// TwinCAT 3 PLC project CNC
// ProgramVersion: 3.1.4020.2
// libraries:
//   Tc2_ControllerToolbox, * (Beckhoff Automation GmbH)
//   Tc2_Standard, * (Beckhoff Automation GmbH)
//   Tc2_System, * (Beckhoff Automation GmbH)
//   Tc2_TcpIp, * (Beckhoff Automation GmbH)
//   Tc2_Utilities, * (Beckhoff Automation GmbH)
//   Tc3_Interfaces, * (Beckhoff Automation GmbH)
//   Tc3_Module, * (Beckhoff Automation GmbH)
//   VisuDialogs, * (System)
// project tree:
//   / ErrorList.TcTLO (not stored), GlobalImagePool.TcGIPO (not stored), GlobalTextList.TcGTLO, PlcTask.TcTTO (not stored), Visualisierungsmanager.TcVMO (not stored), VISU_TASK.TcTTO (not stored)
//   FB_Lib/Conversion/ FB_ConfigAnalog.TcPOU (not stored), FB_Ia.TcPOU (not stored), FB_Qa.TcPOU (not stored), ST_MinMax.TcDUT (not stored)
//   FB_Lib/ErrorAdmin/ FB_ErrorAdmin.TcPOU, ST_ActivatationError.TcDUT, ST_ActivError.TcDUT, ST_CounterError.TcDUT, ST_GestionErreur.TcDUT, ST_InternalError.TcDUT
//   FB_Lib/ErrorAdmin/view/ FB_ErrorViewer.TcPOU, ST_ErrorView.TcDUT
//   FB_Lib/FB_ActionneurSimple/ FB_ActionneurSimple.TcPOU (not stored), ST_Erreur.TcDUT (not stored), ST_ParamActionneur.TcDUT (not stored)
//   FB_Lib/ FB_Etape.TcPOU (not stored), FB_RegulMoteur.TcPOU (not stored)
//   FB_Lib/FB_GestionModes/ FB_Btn.TcPOU (not stored), FB_CycleAuto.TcPOU (not stored), FB_CycleInit.TcPOU (not stored), FB_CycleMan.TcPOU (not stored), FB_MMA.TcPOU (not stored), p_InitVar.TcPOU (not stored)
//   FB_Lib/FB_GestionModes/IO/ ST_IO.TcDUT (not stored), ST_IOInput.TcDUT (not stored), ST_IOInputSimul.TcDUT (not stored), ST_IOOutput.TcDUT (not stored), ST_IOOutputSimul.TcDUT (not stored)
//   FB_Lib/FB_GestionModes/Param/ E_ModeMMA.TcDUT (not stored), ST_Param.TcDUT (not stored), ST_ParamFixed.TcDUT (not stored), ST_ParamRecipe.TcDUT (not stored), ST_ParamStatus.TcDUT (not stored)
//   FB_Lib/TCPIP/ FB_TCP.TcPOU (not stored), ST_Output.TcDUT (not stored), ST_ParamTCP.TcDUT (not stored), ST_TxRx.TcDUT (not stored)
//   GVLs/ GVL.TcGVL
//   POUs/ MAIN.TcPOU
//   VISUs/ VisuAdmin.TcVIS (not stored), Visualization.TcVIS, VisuAuto.TcVIS (not stored), VisuInit.TcVIS (not stored), VisuManual.TcVIS (not stored), VisuMMA.TcVIS (not stored), VisuMotor.TcVIS (not stored), Vi_Alarmes.TcVIS

// ---- FB_Lib/ErrorAdmin/ST_ActivatationError.TcDUT
TYPE ST_ActivatationError :
STRUCT
	/// Set error, starting fbtimer counter
	xError: BOOL;
	/// time before error  
	TimeBeforError: TIME;
	///error level
	iNiveau: BYTE;
	/// error id 
	iId: DINT;
	/// error parameter 
	iIdParam: DINT;
END_STRUCT
END_TYPE

// ---- FB_Lib/ErrorAdmin/ST_ActivError.TcDUT
TYPE ST_ActivError :
STRUCT
	///active error ID
	iId: DINT := 0;
	iParam: DINT := 0;
	///active error parameter
	iIndexOrigine: INT := 0;
	iLevel: BYTE := 0;
END_STRUCT
END_TYPE

// ---- FB_Lib/ErrorAdmin/ST_CounterError.TcDUT
TYPE ST_CounterError :
STRUCT
	iLevel0: INT;
	ilevel1: INT;
	iLevel2: INT;
	iActiv: INT;
	iTotal: INT;
END_STRUCT
END_TYPE

// ---- FB_Lib/ErrorAdmin/ST_GestionErreur.TcDUT
TYPE ST_GestionErreur :
STRUCT
	/// TON 
	fbTime: TON;
	iId: DINT;
	///indique si on a déjà activé l'alarme
	xActivated: BOOL := FALSE;
	/// contient l'adresse dans le tableau d'alarmes actives
	iIdActiv: INT := 0;
END_STRUCT
END_TYPE

// ---- FB_Lib/ErrorAdmin/ST_InternalError.TcDUT
TYPE ST_InternalError :
STRUCT
	xActive: BOOL := FALSE;
	///active error ID
	iId: DINT := 0;
	iParam: DINT := 0;
	sMess: STRING := '';
END_STRUCT
END_TYPE

// ---- FB_Lib/ErrorAdmin/view/ST_ErrorView.TcDUT
TYPE ST_ErrorView :
STRUCT
	id:DINT;
	idparam:DINT;
	sMess:STRING[150];
END_STRUCT
END_TYPE

// ---- GVLs/GVL.TcGVL
VAR_GLOBAL

	fbAct1:FB_ActionneurSimple;	//Act1 corresponds to charging
	fbAct2:FB_ActionneurSimple;	//Act2 corresponds to engraving
	fbAct3:FB_ActionneurSimple;	//Act3 corresponds to tightening
	
	xModeStepForStep :BOOL;
	xNextStep : BOOL;
	
	//pour FB_gestion du mode
	fbMMA:FB_MMA;
	fbCycleAuto:FB_CycleAuto;
	fbCycleInit : FB_CycleInit;
	fbCycleMan : FB_CycleMan;
	
	stParam:ST_Param;
	fbBtn:FB_Btn;
	stIO:ST_IO;
	
	//Tachymetre moteur
	fbMotor : FB_RegulMoteur;
	
	//include TCP_LIB
	fbTCP : FB_TCP;
	
	//
	fbErrorAdmin:FB_ErrorAdmin;//gestion des erreurs, messages
	fbErrorViewer:FB_ErrorViewer;//gestion de l'affichage du tableau
	

	 
END_VAR

// ---- FB_Lib/ErrorAdmin/FB_ErrorAdmin.TcPOU
///*********************************************************************************************************************************************************************
///*{He-Arc}  {Hôtle de ville 7}   {2400 Le Locle}       Phone: ++ 0041 (0)32 930 13 13     Fax: ++ 0041 (0)32 930 13 14         Email: ingenierie@he-arc.ch
///*=======================================================================================================================
///* {Give the complete list of every blocks for a source file with several blocks}
///*
///*=======================================================================================================================
///*Description: Error administration function block
///*
///*=======================================================================================================================
///*Version:        Date:               Author:                           Reason of modification:
///*1.0                   27.11.11         Fabien Golay              Initial Version 
///*1.1                                                                 
///*
///*
///***********************************************************************************************************************************************************************
FUNCTION_BLOCK FB_ErrorAdmin
VAR_OUTPUT
	///in error 
	xInError: BOOL;
	///error level0
	xErrorLevel0: BOOL;
	///error level1 ) 
	xErrorLevel1: BOOL;
	///error level2
	xErrorLevel2: BOOL;
	///tableau des erreurs actuelles
	stActError: ARRAY[0..iMaxErrActiv] OF ST_ActivError;
	///compteur d'erreurs actives
	stCounter: ST_CounterError;
END_VAR
VAR CONSTANT
	iMaxErrActiv: INT := 19;
	iMaxErrId: INT := 1000;
END_VAR
VAR
	stError: ST_ActivatationError;
	stGestion: ARRAY[0..iMaxErrId] OF ST_GestionErreur;
	/// array of  100 timer type TON boMemDeleteError
	iIndex: INT;
	///pour boucle for
	i: INT;
	///si !=0 alors on décompte à chaque mResetIndex (représente 1 fois par cycle automate)
	iInhibSurveille: INT;
END_VAR

///Quittance des erreurs (toutes)
{attribute 'object_name' := 'mAckAll'}
METHOD mAckAll
VAR_INPUT
	iInhibCounter: INT;
END_VAR


(*Reset fbtimer error*)
FOR i:=0 TO iMaxErrActiv DO
	stActError[i].iId:=0;
	stActError[i].iParam:=0;
	stActError[i].iIndexOrigine:=0;
END_FOR
//reset du timer
FOR i:=0 TO iMaxErrId DO
	//stGestion[i].fbTime(in:=FALSE);
	stGestion[i].xActivated:=FALSE;
	stGestion[i].iIdActiv:=0;
END_FOR
(*Reseting error*)
stCounter.iActiv:=0;
stCounter.ilevel0:=0;
stCounter.ilevel1:=0;
stCounter.ilevel2:=0;
xErrorLevel0:=FALSE;				(*on a des erreurs*)
xErrorLevel1:=FALSE;				(*on a des erreurs*)
xErrorLevel2:=FALSE;				(*on a des erreurs*)
xInError:=FALSE;
iInhibSurveille:=iInhibCounter;
END_METHOD

///Quittance d'une seul erreur selon son ID actif
{attribute 'object_name' := 'mAckError'}
METHOD mAckError
VAR_INPUT
	iNoIdActiv: INT;
END_VAR
CASE  stActError[iNoIdActiv].iLevel OF
	1:IF stCounter.ilevel1>0 THEN stCounter.ilevel1:=stCounter.iLevel1+1;END_IF
	2:IF stCounter.ilevel2>0 THEN stCounter.ilevel2:=stCounter.iLevel2+1;END_IF
	ELSE IF stCounter.ilevel0>0 THEN stCounter.ilevel0:=stCounter.iLevel0+1;END_IF
END_CASE

IF stGestion[iNoIdActiv].iIdActiv>=stCounter.iActiv-1
	THEN
		FOR i:=stGestion[iNoIdActiv].iIdActiv TO stCounter.iActiv-1
			DO
				stActError[i]:=stActError[i+1];
				stGestion[iIndex].xActivated:=FALSE;
		END_FOR
END_IF
END_METHOD

///Méthode privée Activation de l'erreur depuis mSurveille
{attribute 'object_name' := 'mActiveError'}
METHOD PRIVATE mActiveError
(*Error level 0=>fatal 1=>warning with validation 2=>warning without validation*)
CASE stError.iNiveau OF
	1:stCounter.ilevel1:=stCounter.iLevel1+1;
	2:stCounter.ilevel2:=stCounter.ilevel2+1;
	ELSE stCounter.ilevel0:=stCounter.ilevel0+1;
END_CASE
xInError:=TRUE;
i:=-1;
REPEAT
	i:=i+1;
	IF stActError[i].iId=0
		THEN
			stActError[i].iId:=stError.iId;
			stActError[i].iParam:=stError.iIdParam;
			stActError[i].iIndexOrigine:=iIndex;
			stActError[i].iLevel:=stError.iNiveau;
			stGestion[iIndex].xActivated:=TRUE;
			stGestion[iIndex].iIdActiv:=i;
			stCounter.iActiv:=stCounter.iActiv+1;
	END_IF
UNTIL (stActError[i].iId=stError.iId AND stActError[i].iParam=stError.iIdParam)
		  OR i=iMaxErrActiv
END_REPEAT;
END_METHOD

///permet d'inhiber une erreur en fonction de son index dans le tableau de surveillance des alarmes
METHOD mInhibeError
VAR_INPUT
	iIndexError: INT;
END_VAR
//réamorcage du timer
IF iInhibSurveille=0
	THEN
		stGestion[iIndexError].fbTime(IN:=FALSE);
		if stGestion[iIndexError].xActivated
			then
				mAckError(stGestion[iIndexError].iIdActiv);
		END_IF
END_IF
END_METHOD

///Efface une erreur de niveau deux dans le tableau des erreurs actives
{attribute 'object_name' := 'mRemoveErrorNv2'}
METHOD PRIVATE mRemoveErrorNv2
IF stCounter.iActiv-1>=stGestion[iIndex].iIdActiv AND stCounter.iActiv<iMaxErrActiv THEN
	FOR i:=stGestion[iIndex].iIdActiv TO stCounter.iActiv-1
	DO
		stActError[i]:=stActError[i+1];
		stGestion[iIndex].xActivated:=FALSE;
		IF stCounter.ilevel2>0
			THEN
				stCounter.ilevel2:=stCounter.ilevel2-1;
		END_IF
		IF stCounter.iActiv>0
			THEN
				stCounter.iActiv:=stCounter.iActiv-1;
		END_IF
	END_FOR
	ELSE 
		stCounter.iActiv:=stCounter.iActiv;
END_IF
END_METHOD

///reset de l'index, doit être éxécuté au début de la tâche automate
{attribute 'object_name' := 'mResetIndex'}
METHOD mResetIndex
stCounter.iTotal:=iIndex-1;
iIndex:=0;
IF iInhibSurveille>0
	THEN
		iInhibSurveille:=iInhibSurveille-1;
END_IF

//contrôle des status d'erreur
xErrorLevel0:=stCounter.iLevel0>0;
xErrorLevel1:=stCounter.iLevel1>0;
xErrorLevel2:=stCounter.iLevel2>0;
//test si plus aucune erreur
xInError:=xErrorLevel0 OR xErrorLevel1 OR xErrorLevel2;
END_METHOD

///ajouter la surveillance pour un ID
{attribute 'object_name' := 'mSetAlaram'}
METHOD mSetAlaram
VAR_INPUT
	/// Set error, starting fbtimer counter
	xError: BOOL;
	///error level
	iNiveau: BYTE;
	/// time before error  
	TimeBeforError: TIME;
	/// error id 
	iId: DINT;
	/// error parameter 
	iIdParam: DINT;
END_VAR

IF iInhibSurveille=0
	THEN
		stError.xError:=xError;
		stError.iNiveau:=iNiveau;
		stError.TimeBeforError:=TimeBeforError;
		stError.iIdParam:=iIdParam;
		stError.iId:=iId;
		mSurveille();
END_IF
END_METHOD

///fonction privée de surveillance des états, pour activation
{attribute 'object_name' := 'mSurveille'}
METHOD PRIVATE mSurveille
(********************************************************************************************************************************************************)
(*											Active fbtimer											 *)
(********************************************************************************************************************************************************)
stGestion[iIndex].fbTime(IN:=stError.xError, PT:= stError.TimeBeforError );
stGestion[iIndex].iId:=stError.iId;
(********************************************************************************************************************************************************)
(*									Write error										 *)
(********************************************************************************************************************************************************)
//si l'activation n'est pas encore faite et que l'alarme apparait
IF stGestion[iIndex].fbTime.Q and not stGestion[iIndex].xActivated
		THEN
		//activation de l'erreur dans le tableau
		mActiveError();
	//test si suppression
	ELSIF stGestion[iIndex].xActivated AND NOT stError.xError
				AND stError.iNiveau=2
		THEN
		//suppression de l'erreur si niveau 2
		 mRemoveErrorNv2();
	END_IF
iIndex:=iIndex+1;
IF iIndex>iMaxErrId THEN
	iIndex:=0;
END_IF
END_METHOD

///retourne la valeur actuel de l'index du tableau de surveillance
PROPERTY pGetIndex : INT
GET

pGetIndex:=iIndex;
END_GET
SET
END_SET
END_PROPERTY

END_FUNCTION_BLOCK

// ---- FB_Lib/ErrorAdmin/view/FB_ErrorViewer.TcPOU
FUNCTION_BLOCK FB_ErrorViewer
VAR_INPUT
	iLangue:INT;
END_VAR
VAR_OUTPUT
	stAcTime:TIMESTRUCT;
	astErrorView: ARRAY [0..iMaxErrActiv]OF ST_ErrorView;
END_VAR
VAR_IN_OUT
	fbErrorAdmin:FB_ErrorAdmin;
END_VAR
VAR CONSTANT
	iMaxErrActiv: INT := 19;
END_VAR
VAR
	fbNTGetTime:NT_GetTime;
	fbEtape:FB_Etape;
	i:INT;
END_VAR

FOR i:=0 TO iMaxErrActiv DO
	IF astErrorView[i].id<>fbErrorAdmin.stActError[i].iId 
		OR astErrorView[i].idparam<>fbErrorAdmin.stActError[i].iParam THEN
		mSetError(i);
	END_IF
END_FOR

fbEtape.mActualisation(FALSE,FALSE);
CASE fbEtape.iNo OF
	0://start read
		fbEtape.piVal:=100;
	100://start
		IF fbNTGetTime.BUSY THEN
			fbEtape.piVal:=110;
		END_IF
	110://wait end 
		IF NOT fbNTGetTime.BUSY
			THEN
				fbEtape.piVal:=120;
		END_IF
	120:IF NOT fbNTGetTime.ERR THEN
			stAcTime:=fbNTGetTime.TIMESTR;
		END_IF
		fbEtape.tTimeQ:=T#1S;
		fbEtape.piVal:=130;
	130:IF fbEtape.xTimeQ THEN
		fbEtape.piVal:=100;
	END_IF
END_CASE

//fonction start dans la boucle
fbNTGetTime(NETID:='',START:=fbEtape.iNo=100,TMOUT:=T#2S);

METHOD mGetActionneurName : STRING
VAR_INPUT
	iIdParam:DINT;
END_VAR
VAR
	sMess:STRING;
END_VAR
CASE iIdParam OF
	1:sMess:='Actionneur 1';
	2:sMess:='Actionneur 2';
	3:sMess:='Actionneur 3';
	ELSE
		sMess:='Actionneur sans nom';
END_CASE

mGetActionneurName:=sMess;
END_METHOD

METHOD mGetErrorMess : STRING
VAR_INPUT
	id:DINT;
	iIdParam:DINT;
END_VAR
VAR
	sMess:STRING;
	iOffset:INT;
END_VAR
CASE iLangue OF
	//fançais
	0:iOffset:=0;
	//allemand
	1:iOffset:=10000;
	//anglais
	2:iOffset:=20000;
	ELSE
		iOffset:=0;
END_CASE
//transformation date et heure, possible également avec Systemtime_to_string()
sMess:=CONCAT(sMess,WORD_TO_STRING(stAcTime.wDay));
sMess:=CONCAT(sMess,'.');
sMess:=CONCAT(sMess,WORD_TO_STRING(stAcTime.wMonth));
sMess:=CONCAT(sMess,'.');
sMess:=CONCAT(sMess,WORD_TO_STRING(stAcTime.wYear));
sMess:=CONCAT(sMess,', ');
sMess:=CONCAT(sMess,WORD_TO_STRING(stAcTime.wHour));
sMess:=CONCAT(sMess,':');
sMess:=CONCAT(sMess,WORD_TO_STRING(stAcTime.wMinute));
sMess:=CONCAT(sMess,':');
sMess:=CONCAT(sMess,WORD_TO_STRING(stAcTime.wSecond));
sMess:=CONCAT(sMess,', ');
mGetErrorMess:=sMess;
CASE id OF
	//français
	0: sMess:='Erreur 0';
	1: sMess:='Erreur 1';
	3: sMess:='Arrêt d urgence';
	10:sMess:='Autorisation refusée pour action rentrer';
		
	11:sMess:='Autorisation refusée pour action sortir';
		sMess:=CONCAT(sMess,', ');
		sMess:=CONCAT(sMess,mGetActionneurName(iIdParam));
	20:sMess:='Erreur de timeout rentre';
		sMess:=CONCAT(sMess,', ');
		sMess:=CONCAT(sMess,mGetActionneurName(iIdParam));
	21:sMess:='Erreur de Moteur';
		sMess:=CONCAT(sMess,', ');
		sMess:=CONCAT(sMess,mGetActionneurName(iIdParam));
	30:sMess:='Erreur de Pression air';
		sMess:=CONCAT(sMess,', ');
		sMess:=CONCAT(sMess,mGetActionneurName(iIdParam));
	31:sMess:='Double consignes, xSetSort=1 et xSetRentre=1';
		sMess:=CONCAT(sMess,', ');
		sMess:=CONCAT(sMess,mGetActionneurName(iIdParam));
	40:sMess:='Erreur perte signal FDC rentre';
		sMess:=CONCAT(sMess,', ');
		sMess:=CONCAT(sMess,mGetActionneurName(iIdParam));
	41:sMess:='Erreur perte signal FDC sort';
		sMess:=CONCAT(sMess,', ');
		sMess:=CONCAT(sMess,mGetActionneurName(iIdParam));
	//allemand
	10000: sMess:='Erreur 0';
	10001: sMess:='Erreur 1';
	//anglais
	20000: sMess:='Erreur 0';
	20001: sMess:='Erreur 1';
	ELSE
		sMess:='Le message n existe pas';
END_CASE

mGetErrorMess:=concat(mGetErrorMess,sMess);
END_METHOD

METHOD PRIVATE mSetError : BOOL
VAR_INPUT
	i:INT;
END_VAR
astErrorView[i].id:=fbErrorAdmin.stActError[i].iId;
astErrorView[i].idparam:=fbErrorAdmin.stActError[i].iParam;
IF astErrorView[i].id=0 THEN
		//vider le message
		astErrorView[i].sMess:='';
	ELSE
		//lecture du message d'erreur
		astErrorView[i].sMess:=mGetErrorMess(astErrorView[i].id, astErrorView[i].idparam);
END_IF


//gestion du fichier de log
//mLogError();
END_METHOD

END_FUNCTION_BLOCK

// ---- POUs/MAIN.TcPOU
PROGRAM MAIN
VAR
	xSetError:BOOL;
	iNiveau:BYTE:=0;
	TimeBeforError: TIME := T#100MS;
	iId:INT:=1;
	iIdParam:INT := 100;
END_VAR

//initialisation du gestionnaire d'alarmes
fbErrorAdmin.mResetIndex();
//Refresh du viewer d'alarmes
fbErrorViewer(fbErrorAdmin:=fbErrorAdmin);
//quittance des erreurs dans FB_MMA, iEtape=810
//exemple d'ajout d'une erreur
fbErrorAdmin.mSetAlaram(xError :=xSetError,
						iNiveau:=iNiveau,
						TimeBeforError:=TimeBeforError,
						iId:=iId,
						iIdParam:=iIdParam);





//******************************************
//cyclic call of all needed FB
//******************************************

fbAct1();	//Act1 corresponds to charging
fbAct2();	//Act2 corresponds to engraving
fbAct3();	//Act3 corresponds to tightening
fbMMA();

//copy physical Inputs in fbBtn
fbBtn.xAru:=stio.stIn.IxAruIO;
fbBtn.xReset:=stio.stIn.xResetIO OR NOT stio.stIn.xAirPressureOk;
fbBtn.xStart:=stio.stIn.xStartIO;
fbBtn.xStop:=stio.stIn.xStopIO;
fbBtn.xAirPressureOk:=stio.stIn.xAirPressureOk;
fbBtn.xManualAct1GoIn:=stio.stIn.xManualAct1GoIn;
fbBtn.xManualAct1GoOut:=stio.stIn.xManualAct1GoOut;
fbBtn.xManualAct2GoIn:=stio.stIn.xManualAct2GoIn;
fbBtn.xManualAct2GoOut:=stio.stIn.xManualAct2GoOut;
fbBtn.xManualAct3GoIn:=stio.stIn.xManualAct3GoIn;
fbBtn.xManualAct3GoOut:=stio.stIn.xManualAct3GoOut;
fbBtn.xManualCNCMotorTurnOn:=stio.stIn.xManualCNCMotorTurnOn;
fbBtn.xManualCNCMotorTurnOff:=stio.stIn.xManualCNCMotorTurnOff;
fbBtn.xEmulateTCPConnection:=stio.stIn.xEmulateTCPConnection;
fbBtn.xManualSendTrig:=stio.stIn.xManualSendTrig;
fbBtn.xManualSendCheck:=stio.stIn.xManualSendCheck;
fbBtn.xManualSendGetres:=stio.stIn.xManualSendGetres;
//and now call it
fbBtn();

//stParam
//check for active errors
fbErrorAdmin.mSetAlaram(xError :=fbAct1.stError.xState,
						iNiveau:=0,
						TimeBeforError:=T#100MS,
						iId:=0,
						iIdParam:=1);
fbErrorAdmin.mSetAlaram(xError :=fbAct2.stError.xState,
						iNiveau:=0,
						TimeBeforError:=T#100MS,
						iId:=0,
						iIdParam:=2);
fbErrorAdmin.mSetAlaram(xError :=fbAct3.stError.xState,
						iNiveau:=0,
						TimeBeforError:=T#100MS,
						iId:=0,
						iIdParam:=2);
fbErrorAdmin.mSetAlaram(xError :=fbMotor.xError,
						iNiveau:=0,
						TimeBeforError:=T#100MS,
						iId:=21,
						iIdParam:=0);
fbErrorAdmin.mSetAlaram(xError :=fbBtn.xAirPressureOk,
						iNiveau:=0,
						TimeBeforError:=T#100MS,
						iId:=30,
						iIdParam:=0);



//******
IF (fbAct1.stError.xState) THEN
	stParam.stStatus.xErreur:=TRUE;
	stParam.stStatus.iId:=fbAct1.stError.iId;
	
ELSIF (fbAct2.stError.xState) THEN
	stParam.stStatus.xErreur:=TRUE;
	stParam.stStatus.iId:=fbAct2.stError.iId;
	
ELSIF (fbAct3.stError.xState) THEN
	stParam.stStatus.xErreur:=TRUE;
	stParam.stStatus.iId:=fbAct3.stError.iId;
ELSIF (fbCycleAuto.xError) THEN
	stParam.stStatus.xErreur:=TRUE;
	stParam.stStatus.iId:=fbCycleAuto.iId;
ELSIF (fbMotor.xError) THEN
	stParam.stStatus.xErreur:=TRUE;
	stParam.stStatus.iId:=fbMotor.iErrorID;
ELSIF (fbTCP.OutputGlobal.xError) THEN
	stParam.stStatus.xErreur:=TRUE;
	stParam.stStatus.iId:=fbTCP.OutPutGlobal.nErrID;
ELSIF NOT fbBtn.xAirPressureOk THEN
	stParam.stStatus.xErreur:=TRUE;
	stParam.stStatus.iId:=1;
ELSE
	//clear the error State. Do not clear the last error Message to have some kind of error history
	stParam.stStatus.xErreur:=FALSE;
END_IF

//call auto mode and give over the needed parameters
fbCycleAuto.xStart:=fbMMA.iEtape=350;
fbCycleAuto.xStop:= fbMMA.iEtape=390;
fbCycleAuto.xReset:= fbMMA.iEtape=810 OR fbMMA.iEtape=910;
fbCycleAuto();

//call Init mode and give over the needed parameters
fbCycleInit.xStart:=(fbMMA.iEtape=110 OR fbMMA.iEtape=340);
fbCycleInit.xStop:= NOT (fbMMA.iEtape=111 OR fbMMA.iEtape=341);
fbCycleInit.xReset:= fbMMA.iEtape=810 OR fbMMA.iEtape=910;
fbCycleInit();
	
//call Manual mode and give over the needed parameters
fbCycleMan.xStart:= fbMMA.iEtape=210;
fbCycleMan.xStop:=  fbMMa.iEtape<>210;
fbCycleMan();

//call Motor Controller
fbMotor.Consigne:=stIO.stIn.lSetSpeedMotor;
fbMotor.fbConvertTachoToNumSpeed.IaEntree:=stio.stIn.lTachoValue;
fbMotor.xDirection:=stio.stIn.xMotorDirection;
fbMotor();
stio.stOut.lMotorOut:=fbMotor.fbConvertNumToMotorOut.QaSortie;

//call TCP Block
fbTCP();

//******************************************
//Output actions
//******************************************

//activate Lamp1
stIo.stOut.QxLampeRed:=fbCycleAuto.iEtape<800 AND fbCycleAuto.iEtape>0;

//actuator movement autorize only if not in ARU
fbAct1.xAutorizeIn:=fbBtn.xAru;
fbAct1.xAutorizeOut:=fbBtn.xAru;
fbAct2.xAutorizeIn:=fbBtn.xAru;
fbAct2.xAutorizeOut:=fbBtn.xAru;
fbAct3.xAutorizeIn:=fbBtn.xAru;
fbAct3.xAutorizeOut:=fbBtn.xAru;

//move in and out each actuator
fbAct1.xInGoOut:=fbCycleAuto.iEtape=130 OR fbCycleMan.iEtape=202;
fbAct2.xInGoOut:=fbCycleAuto.iEtape=160 OR fbCycleMan.iEtape=204;
fbAct3.xInGoOut:=fbCycleAuto.iEtape=140 OR fbCycleMan.iEtape=206;

fbAct3.xInGoIn:=fbCycleAuto.iEtape=180 OR fbCycleAuto.iEtape=800 OR fbCycleInit.iEtape=100 OR fbCycleMan.iEtape=205;
fbAct2.xInGoIn:=fbCycleAuto.iEtape=170 OR fbCycleAuto.iEtape=800 OR fbCycleInit.iEtape=100 OR fbCycleMan.iEtape=203;
fbAct1.xInGoIn:=fbCycleAuto.iEtape=180 OR fbCycleAuto.iEtape=800 OR fbCycleInit.iEtape=100 OR fbCycleMan.iEtape=201;

//Motor
IF(fbCycleAuto.iEtape=140 OR fbCycleMan.iEtape=207) THEN
	fbMotor.xOnOff:=TRUE;
END_IF
IF(fbCycleAuto.iEtape=170 OR fbCycleInit.iEtape=100 OR fbCycleMan.iEtape=208 OR fbCycleAuto.iEtape=800 OR fbMMA.iEtape=910 OR fbMMA.iEtape=810) THEN
	fbMotor.xOnOff:=FALSE;
END_IF
//Reset fbMotor
fbMotor.xReset:=fbMMA.iEtape=810;
//Motor Direction Output
stio.stOut.QxMotorDirection:=stio.stIn.xMotorDirection;

//Reset des Actionneurs avan le init
fbAct1.xReset:=fbCycleInit.iEtape=99 OR fbMMA.iEtape=810;
fbAct2.xReset:=fbCycleInit.iEtape=99 OR fbMMA.iEtape=810;
fbAct3.xReset:=fbCycleInit.iEtape=99 OR fbMMA.iEtape=810;

//Reset de la connexion TCIP
fbTCP.xForceDisconnect:=fbMMA.iEtape=810 OR fbCycleInit.iEtape=100;
IF fbCycleInit.iEtape=102 THEN
	fbTCP.xEnable:=TRUE;
END_IF

//TCP send data
IF fbCycleAuto.iEtape=111 OR fbCycleAuto.iEtape=190 OR fbCycleMan.iEtape=209 THEN
	fbTCP.TxRx.sSend:='TRIG';
END_IF
IF fbCycleAuto.iEtape=192 OR fbCycleMan.iEtape=210 THEN
	fbTCP.TxRx.sSend:='GETRES';
END_IF
IF fbCycleAuto.iEtape=113 OR fbCycleMan.iEtape=211 THEN
	fbTCP.TxRx.sSend:='CHECK';
END_IF

//clear received string
IF fbCycleAuto.iEtape=113 OR fbCycleAuto.iEtape=800 OR fbCycleAuto.iEtape=130 OR fbCycleAuto.iEtape=192 OR fbCycleAuto.iEtape=200
OR fbMMA.iEtape=810 OR fbCycleInit.iEtape=100 THEN
	fbTCP.TxRx.sReceived:='';
END_IF

END_PROGRAM

// ---- GlobalTextList.TcGTLO
TEXTLIST GlobalTextList
  58 = '%d'
  37 = '%i'
  3 = '%s'
  60 = 'Act1'
  62 = 'Act2'
  61 = 'Act3'
  15 = 'Actionneur 1' | fr: 'Actionneur 1' | de: 'Aktor 1' | en: 'Actuator 1'
  16 = 'Actionneur 2' | fr: 'Actionneur 2' | de: 'Aktor 2' | en: 'Actuator 2'
  17 = 'Actionneur 3' | fr: 'Actionneur 3' | de: 'Aktor 3' | en: 'Actuator 3'
  40 = 'Admin'
  67 = 'ADMIN'
  127 = 'Air pressure emulator'
  8 = 'ARU' | fr: 'ARU' | de: 'NOT-Aus' | en: 'emergency Stop'
  93 = 'ARU - when there is no hardwarebutton present' | fr: 'ARU - seulement si il y a pas de Bouton Hardware' | de: 'NOT-Aus - nur wenn es kein Hardware-Button gibt' | en: 'emergency Stop - only when there is no Hardware Button'
  71 = 'AUTOMATIC' | fr: 'AUTOMATIQUE' | de: 'AUTOMATISCH'
  126 = 'Camera Control'
  53 = 'Charge' | fr: 'Charge' | de: 'Laden' | en: 'Load'
  96 = 'Connected to Server' | fr: 'Connecté aux Serveur' | de: 'Verbunden mit Serveur'
  25 = 'Consigne: %.2f' | fr: 'Consigne: %.2f' | de: 'Soll-Wert: %.2f' | en: 'Setpoint: %.2f'
  0 = 'Cycle Init' | fr: 'CYCLE INITIALISATION' | de: 'INITIALISIERUNGSZYKLUS' | en: 'INITIALISATION CYCLE'
  5 = 'Cycle Man' | fr: 'CYCLE MANUEL' | de: 'MANUELLER ZYKLUS' | en: 'MANUAL CYCLE'
  92 = 'd: %s'
  63 = 'Direction' | fr: 'Sens de rotation' | de: 'Drehrichtung' | en: 'Direction'
  76 = 'Disable Sensor In - Out' | fr: 'Désactiver Capteur In-Out' | de: 'In-Out Sensor deaktivieren' | en: 'Disable Sensor In-Out'
  114 = 'Do next step if Pas-a-Pas is enabled' | fr: 'Faire le prochain pas si Pas-a-Pas est allumée' | de: 'Nächster Schritt wenn Schritt-für-Schritt aktiviert ist' | en: 'Do next step if Step-for-Step is turned on'
  113 = 'Do Step' | fr: 'Faire un pas' | de: 'Schritt' | en: 'Do Step'
  90 = 'e: %s'
  97 = 'Enabled' | fr: 'Activé' | de: 'Aktiviert'
  41 = 'english' | fr: 'Anglais' | de: 'Englisch' | en: 'English'
  78 = 'ErrID: %d'
  7 = 'Error' | fr: 'Erreur' | de: 'Fehler' | en: 'Error'
  33 = 'fbConfig.lrTemp : %.2f'
  36 = 'fbConfig.lrValInc : %.2f'
  32 = 'fbConfig.udiNbreIncBus : %i'
  105 = 'fbMotor.fbMotor.fbConvertNumToMotorOut.QaSortie'
  98 = 'Force Disconnect' | de: 'Zwangs-Trennen'
  19 = 'french' | fr: 'Francais' | de: 'Französisch' | en: 'French'
  43 = 'Gain : %.2f'
  20 = 'german' | fr: 'Allemand' | de: 'Deutsch' | en: 'German'
  65 = 'go back' | fr: 'retour...' | de: 'zurück...' | en: 'go back...'
  66 = 'go back...' | fr: 'retour...' | de: 'zurück...' | en: 'go back...'
  22 = 'Going in' | fr: 'rétracter' | de: 'ein-fahren' | en: 'retract'
  21 = 'Going out' | fr: 'étendre' | de: 'aus-fahren' | en: 'extend'
  91 = 'h: %s'
  48 = 'ID: %d'
  132 = 'iId: %d'
  133 = 'iIdParam: %d'
  130 = 'iNiveau: %d'
  102 = 'Ir Ecart : %.5f'
  103 = 'Ir Tension: %.2f'
  2 = 'LANGUAGE' | fr: 'LANGUE' | de: 'SPRACHE' | en: 'LANGUAGE'
  115 = 'Login' | fr: 'Connecter' | de: 'Einloggen'
  119 = 'login as another user' | fr: 'Login comme autre utilisateur' | de: 'Als anderen Benutzer einloggen'
  116 = 'Logout' | fr: 'Déconnecter' | de: 'Ausloggen'
  34 = 'lrEcart : %.5f'
  35 = 'lrTension : %.2f'
  4 = 'MAIN' | fr: 'PRINCIPAL' | de: 'HAUPTSEITE' | en: 'MAIN'
  109 = 'MAIN.fbCycleInit.fbEtape.sMess'
  108 = 'MAIN.fbCycleInit.iEtape'
  106 = 'MAIN.fbCycleMan.fbEtape.sMess'
  107 = 'MAIN.fbCycleMan.iEtape'
  6 = 'MMA'
  13 = 'Mode Auto'
  12 = 'Mode Init'
  14 = 'Mode Manual'
  112 = 'Mode Pas-a-Pas'
  55 = 'Motor' | fr: 'Moteur' | de: 'Motor' | en: 'Motor'
  59 = 'MOTOR' | fr: 'MOTEUR' | de: 'MOTOR' | en: 'MOTOR'
  89 = 'NetID: %s'
  39 = 'None'
  110 = 'Num Output: %d'
  111 = 'Num Output: %i'
  73 = 'Number produced: %d' | fr: 'Nombre produits: %d' | de: 'Anzahl Produziert: %d' | en: 'Number produced: %d'
  75 = 'On            Off'
  68 = 'Open Admin Page' | fr: 'Page administrateur...' | de: 'Admin-Seite' | en: 'Admin Page...'
  64 = 'open more...' | fr: "plus d'info..." | de: 'mehr...' | en: 'open more...'
  46 = 'Operator'
  47 = 'Operator - Service - Admin'
  120 = 'Please login as another user' | fr: 'Veuillez utiliser un autre identifiant' | de: 'Bitte mit anderen Benutzerkennung einloggen'
  104 = 'Qa Sortie : %d'
  101 = 'Qa Sortie : %i'
  38 = 'QaSortie : %2.5f'
  42 = 'QaSortie : %2.5f tr/min'
  31 = 'QaSortie : %i'
  100 = 'QASortie: %i'
  70 = 'Ready' | fr: 'Pret' | de: 'Bereit' | en: 'Ready'
  57 = 'RealSpeed: %d'
  85 = 'Received Data: %s'
  80 = 'Remote IP-Adress: %s'
  81 = 'Remote Port: %d'
  72 = 'Remote Socket: %d'
  10 = 'Rentre       Sort'
  11 = 'Rentre      Sort'
  9 = 'Rentre     Sort'
  49 = 'Reset'
  69 = 'Running' | fr: 'Marche' | de: 'Betrieb' | en: 'Running'
  82 = 'Send Data: %s'
  45 = 'Service'
  1 = 'SetSpeed of Motor: %.2f'
  99 = 'SetSpeed of Motor: %i'
  56 = 'SetSpeed: %d'
  23 = 'Start'
  26 = 'stConfigBus.uiNbBits: %i'
  24 = 'Stop'
  27 = 'stTension.lrMax : %.2f'
  28 = 'stTension.lrMin : %.2f'
  29 = 'stValeur.lrMax : %.2f'
  30 = 'stValeur.lrMin : %.2f'
  129 = "Tableau d'affichage des alarmes"
  128 = 'Tableau de gestion des alarmes'
  18 = 'TachoInput: %.2f'
  95 = 'TCP Busy'
  123 = 'TCP Send'
  54 = 'Tighten' | fr: 'Serrage' | de: 'Spannen' | en: 'Tighten'
  131 = 'TimeBeforErr: %d'
  125 = 'TRIG    CHECK   GETRES'
  124 = 'TRIG CHECK GETRES'
  117 = 'User'
  121 = 'USER' | fr: 'UTILISATEUR' | de: 'BENUTZER'
  122 = 'User Settings' | fr: 'Param. Utilisateur' | de: 'Benutzer Einst.'
  44 = 'WriteSpeed: %d'
  74 = 'xBusy'
  83 = 'xConnected'
  86 = 'xConnectedCognex'
  94 = 'xConnectedCognex Native'
  51 = 'xEnable'
  87 = 'xEnableCognexMode'
  88 = 'xEnableEmulateTCP'
  77 = 'xError'
  84 = 'xForceDisconnect'
  79 = 'xSend'
  50 = 'xVonnected'
  118 = 'You are not allowed to see this page' | fr: 'Yous avez pas le droit de voir cette page' | de: 'Sie haben nicht die erforderlichen Recte diese Seite einzusehen'
  52 = 'Z-Axis' | fr: 'Axe Z' | de: 'Z-Achse' | en: 'Z-Axis'
END_TEXTLIST

// ---- VISUs/Visualization.TcVIS
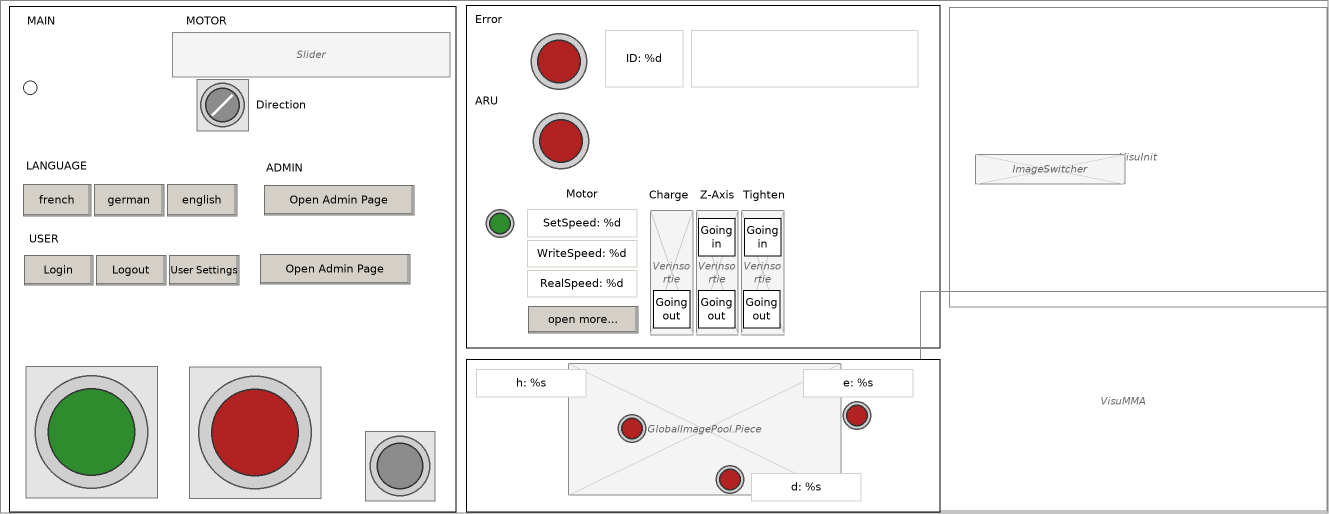
VISUALIZATION Visualization  // 1329x514
    Rectangle (466,5 474x343)
    Rectangle (9,6 447x506)
    Label (24,6 80x30), "MAIN"
    Lamp1 (527,108 68x66), variable: fbBtn.xAru=0, style: Lamp-Lamp1-Red
    Label (472,87 87x28), "ARU"
    RadioButton (21,39 150x97), variable: stParam.stStatus.eMMA
        Areas[0]: Text=Mode Init
        Areas[1]: Text=Mode Auto
        Areas[2]: Text=Mode Manual
    Frame (949,7 378x300), frame switch variable: stParam.stStatus.eMMA
        shows VisuInit()
        shows VisuAuto()
        shows VisuManual()
        shows VisuMMA()
    Frame (920,291 407x220)
        shows VisuMMA()
    Lamp1 (526,27 66x69), variable: stParam.stStatus.xErreur, style: Lamp-Lamp1-Red
    Label (472,5 55x29), "Error"
    Textfield (691,30 227x57), text variable: stParam.stStatus.sMessage, text list: 'ErrorList', text index: stParam.stStatus.iId
    Textfield (605,30 78x57), "ID: %d", text variable: stParam.stStatus.iId
    PushSwitch (24,366 135x132), tooltip "Start", variable: stIO.stIn.xStartIO, behaviour: TAP, style: Switch-PushSwitch-Green
    PushSwitch (189,364 132x137), tooltip "Stop", variable: stIO.stIn.xStopIO, invisible if: fbMMA.iEtape<>350, behaviour: TAP, style: Switch-PushSwitch-Red
    PushSwitch (365,431 70x70), tooltip "Reset", variable: stIO.stIn.xResetIO, behaviour: TAP, style: Switch-PushSwitch-Gray
    Slider (172,32 278x45), variable: stIO.stIn.lSetSpeedMotor, scale 100..1500
    Label (183,6 80x30), "MOTOR"
    Label (253,90 117x30), "Direction"
    RotarySwitch (195,79 55x52), variable: stIO.stIn.xMotorDirection, behaviour: TOGGLE, style: Switch-RotarySwitch-Gray
    Button (264,185 150x30), "Open Admin Page"
        OnMouseClick: change screen: VisuAdmin
    Label (263,153 80x30), "ADMIN"
    Button (23,184 68x32), "french"
        OnMouseClick: ChangeLanguage ChangeLanguage=fr
    Label (23,151 80x30), "LANGUAGE"
    Button (94,184 70x32), "german"
        OnMouseClick: ChangeLanguage ChangeLanguage=de
    Button (167,184 70x32), "english"
        OnMouseClick: ChangeLanguage ChangeLanguage=en
    Label (724,180 80x30), "Tighten"
    Label (629,180 80x30), "Charge"
    Label (677,180 80x30), "Z-Axis"
    Image (741,210 43x125), invisible if: fbAct3.xInInPos=0, image: Verinrentree
    Image (696,210 42x125), invisible if: fbAct2.xInInPos=0, image: Verinrentree
    Image (650,210 43x125), invisible if: fbAct1.xInInPos=0, image: Verinrentree
    Image (650,210 43x125), invisible if: fbAct1.xInOutPos=0, image: Verinsortie
    Image (696,210 42x125), invisible if: fbAct2.xInOutPos=0, image: Verinsortie
    Image (741,210 43x125), invisible if: fbAct3.xInOutPos=0, image: Verinsortie
    Rectangle (743,290 37x38), "Going out", invisible if: fbAct3.xGoingOutNow=0
    Rectangle (698,290 37x38), "Going out", invisible if: fbAct2.xGoingOutNow=0
    Rectangle (653,290 37x38), "Going out", invisible if: fbAct1.xGoingOutNow=0
    Rectangle (744,218 37x38), "Going in", invisible if: fbAct3.xGoingInNow=0
    Rectangle (698,218 37x38), "Going in", invisible if: fbAct2.xGoingInNow=0
    Label (527,179 110x30), "Motor"
    Lamp1 (482,207 36x33), variable: fbMotor.xOnOff, style: Lamp-Lamp1-Green
    Textfield (527,209 110x28), "SetSpeed: %d", text variable: fbMotor.Consigne
    Textfield (527,270 110x27), "RealSpeed: %d", text variable: fbMotor.fbConvertTachoToNumSpeed.lrValeur
    Button (528,306 110x27), "open more..."
        OnMouseClick: change screen: VisuMotor
    Textfield (527,240 110x27), "WriteSpeed: %d", text variable: fbMotor.fbConvertNumToMotorOut.lrConsigne
    Rectangle (466,359 474x153)
    Image (568,363 273x132), image: GlobalImagePool.Piece
    Textfield (803,369 110x28), "e: %s", text variable: fbTCP.OutputGlobal.Resulte
        p3092690914: fbTCP.OutputGlobal.Boole
    Textfield (476,369 110x28), "h: %s", text variable: fbTCP.OutputGlobal.Resulth
    Textfield (751,473 110x28), "d: %s", text variable: fbTCP.OutputGlobal.Resultd
    Lamp1 (614,412 36x33), variable: fbTCP.OutputGlobal.Boolh=0, style: Lamp-Lamp1-Red
    Lamp1 (839,399 36x33), variable: fbTCP.OutputGlobal.Boole=0, style: Lamp-Lamp1-Red
    Lamp1 (712,463 36x33), variable: fbTCP.OutputGlobal.Boold=0, style: Lamp-Lamp1-Red
    ImageSwitcher (975,154 150x30), behaviour: TOGGLE
    Button (382,261 1x2)
    Button (24,255 69x30), "Login"
        OnMouseClick: VisuUserMgmt Type=Login
    Button (96,255 70x30), "Logout"
        OnMouseClick: VisuUserMgmt Type=Logout
    Label (26,224 80x30), "USER"
    Button (169,255 70x30), "User Settings"
        OnMouseClick: VisuUserMgmt Type=OpenUserConfiguration
    Button (260,254 150x30), "Open Admin Page"
        OnMouseClick: change screen: Vi_Alarmes
END_VISUALIZATION

// ---- VISUs/Vi_Alarmes.TcVIS
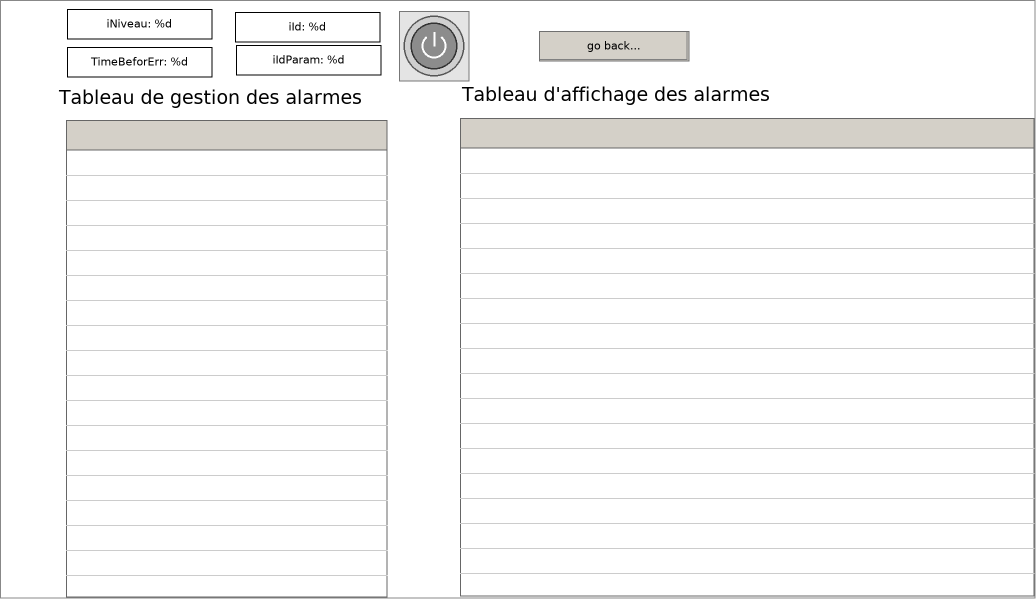
VISUALIZATION Vi_Alarmes  // 1036x599
    Table (66,120 321x477), data array: fbErrorAdmin.stActError
        p3854506369: fbErrorAdmin.stActError[INDEX].iId
        p1892666644: fbErrorAdmin.stActError[INDEX].iParam
        p338671338: fbErrorAdmin.stActError[INDEX].iIndexOrigine
        p2170511999: fbErrorAdmin.stActError[INDEX].iLevel
    Label (56,77 342x41), "Tableau de gestion des alarmes"
    Label (459,74 342x41), "Tableau d'affichage des alarmes"
    Table (460,118 574x478), data array: fbErrorViewer.astErrorView
        p3854506369: fbErrorViewer.astErrorView[INDEX].id
        p1892666644: fbErrorViewer.astErrorView[INDEX].idparam
        p338671338: fbErrorViewer.astErrorView[INDEX].sMess
    Rectangle (67,9 145x30), "iNiveau: %d", text variable: MAIN.iNiveau
        OnMouseClick: write the text variable via Default
    Rectangle (67,47 145x30), "TimeBeforErr: %d", text variable: MAIN.TimeBeforError
        OnMouseClick: write the text variable via Default
    Rectangle (235,12 145x30), "iId: %d", text variable: MAIN.iId
        OnMouseClick: write the text variable via Default
    Rectangle (236,45 145x30), "iIdParam: %d", text variable: MAIN.iIdParam
        OnMouseClick: write the text variable via Default
    PowerSwitch (399,11 70x70), variable: MAIN.xSetError, behaviour: TAP, style: Switch-PowerSwitch-Gray
    Button (539,31 150x30), "go back..."
        OnMouseClick: change screen: Visualization
END_VISUALIZATION
